FUNCTION_BLOCK INTERNAL FB_AlarmManager_Tests EXTENDS FB_TestSuite
VAR
	_dateTime	: ZigaLibs_Core.FB_LocalSystemTimeProvider;
	_alarmManager : FB_AlarmManager(
		enable := TRUE, // [BOOL] - Enables alarm generation
		logger := 0, // [REFERENCE TO ZigaLibs_Core.I_LoggerEx] - optional, logger.
		timeProvider := _dateTime); //[ZigaLibs_Core.I_LocalSystemTimeProvider] - required, date time provider.
END_VAR

_dateTime();
Test00_RegisterAlarms();
Test01_ActivateNewAlarm_ExpectUnacknowledgedActiveAlarm();
Test02_AcknowledgeActiveAlarm_ExpectActiveAcknowledged();
Test03_ActivateExistingAlarm_ExpectSameActiveAlarmCount();
Test04_DeactivateAlarm_ExpectNotActiveAcknowledged();
Test05_AcknowlidgeInactiveAlarm_ExpectAcknowledgedNotActive();
Test06_DisableManager_ExpectNoActiveAlarms();
Test07_AcknowledgeAllAlarms_ExpectActiveAlarmsUnchanged();
Test08_ActivateByName();
Test09_DeactivateByName();
Test10_AcknowledgeByName();
Test11_GetAlarmByName();
Test12_GetAlarmById();
Test13_ActivateById();
Test14_DeactivateById();
Test15_AcknowledgeById();
Test16_TimeInfos();
Test17_RaiseUnexisitngAlarm_ExpectNoNewAlarmsActive();
Test18_DeleteAlarm_ExpectPreviousAlarmsStillExist();
Test19_DeleteUnexistingAlarm_ExpectNoChangesToExistingAlarms();
Test20_DeleteAll();

METHOD Test00_RegisterAlarms
VAR_INPUT
END_VAR

VAR
	addAlarmIndex	: T_ArrayIndexer;
	alarm			: ST_AlarmInfo;
END_VAR
IF TcUnit.TEST_ORDERED('Test00_RegisterAlarms') THEN
	AssertEquals_UDINT(
		Actual := _alarmManager.RegisteredAlarmsCount,
		Expected := 0,
		Message := 'Before registering any alarms, the Registered count should be 0.');
	
	FOR addAlarmIndex := 1 TO 100 BY 1 DO
		AssertTrue(
			Condition := _alarmManager.RegisterAlarm(
				Id := addAlarmIndex,
				Message := Tc2_Standard.CONCAT('Alarm message', TO_STRING(addAlarmIndex)),
				Name := Tc2_Standard.CONCAT('Alarm name', TO_STRING(addAlarmIndex)),
				Level := E_AlarmLevel.INFO),
			Message := 'Registering alarm failed.');
			
		AssertEquals_UDINT(
			Actual := _alarmManager.RegisteredAlarmsCount,
			Expected := DINT_TO_UDINT(addAlarmIndex),
			Message := 'Registered alarm count is incorrect.');
			
		alarm := _alarmManager.GetAlarmById(nID := addAlarmIndex);
		AssertTrue(
			Condition := alarm.IsAcknowledged,
			Message := 'Newly registered alarm should be acknowledged by default, when created.');
	END_FOR
	
	AssertFalse(
		Condition := _alarmManager.RegisterAlarm(
			Id := 22,
			Message := CONCAT('Alarm message', TO_STRING(addAlarmIndex - 1)),
			Name := CONCAT('Alarm name', TO_STRING(addAlarmIndex - 1)),
			Level := E_AlarmLevel.INFO),
		Message := 'Registering an alarm with an existing id should not be possible.');
	
		
	TcUnit.TEST_FINISHED();
END_IF
END_METHOD

METHOD Test01_ActivateNewAlarm_ExpectUnacknowledgedActiveAlarm
VAR_INPUT
END_VAR

VAR
	currentAlarm	: ST_AlarmInfo;
END_VAR
IF TcUnit.TEST_ORDERED('Test01_ActivateNewAlarm_ExpectUnacknowledgedActiveAlarm') THEN
	_alarmManager.RaiseAlarmById(10);
	currentAlarm := _alarmManager.GetAlarmById(10);
	
	AssertEquals_BOOL(
		Actual := currentAlarm.IsActive,
		Expected := TRUE,
		Message := 'Alarm activation failed.');
		
	AssertEquals_BOOL(
		Actual := currentAlarm.IsAcknowledged,
		Expected := FALSE,
		Message := 'Newly activated alarm should not be acknowledged.');	
	
		
	AssertEquals_UINT(
		Actual := _alarmManager.ActiveAlarmsCount,
		Expected := 1,
		Message := 'Active alarm count is incorrect.');
	
	AssertEquals_UINT(
		Actual := _alarmManager.UnacknowledgedAlarmsCount,
		Expected := 1,
		Message := 'Unacknowledged alarm count is incorrect.');
		
	TcUnit.TEST_FINISHED();
END_IF
END_METHOD

METHOD Test02_AcknowledgeActiveAlarm_ExpectActiveAcknowledged
VAR_INPUT
END_VAR
IF TcUnit.TEST_ORDERED('Test02_AcknowledgeActiveAlarm_ExpectActiveAcknowledged') THEN

	_alarmManager.AcknowledgeAlarmById(10);
	
	AssertEquals_BOOL(
		Actual := _alarmManager.GetAlarmById(10).IsActive,
		Expected := TRUE,
		Message := 'Alarm activation failed.');
		
	AssertEquals_BOOL(
		Actual := _alarmManager.GetAlarmById(10).IsAcknowledged,
		Expected := TRUE,
		Message := 'Acknowlidging active alarm failed.');	
	
	TcUnit.TEST_FINISHED();
END_IF
END_METHOD

METHOD Test03_ActivateExistingAlarm_ExpectSameActiveAlarmCount
VAR_INPUT
END_VAR
IF TcUnit.TEST_ORDERED('Test03_ActivateExistingAlarm_ExpectSameActiveAlarmCount') THEN
	_alarmManager.RaiseAlarmById(10);	
	AssertEquals_BOOL(
		Actual := _alarmManager.GetAlarmById(10).IsActive,
		Expected := TRUE,
		Message := 'Alarm activation failed.');
		
	AssertEquals_BOOL(
		Actual := _alarmManager.GetAlarmById(10).IsAcknowledged,
		Expected := TRUE,
		Message := 'Already acknowledged alarm should not be acknowledged when activating the alarm while it is already active.');	
	
		
	AssertEquals_UINT(
		Actual := _alarmManager.ActiveAlarmsCount,
		Expected := 1,
		Message := 'Active alarm count is incorrect.');
	
	AssertEquals_UINT(
		Actual := _alarmManager.UnacknowledgedAlarmsCount,
		Expected := 0,
		Message := 'Activating acknowledged and already active alarm should not cause the alarm to be unacknowledged..');
		
	TcUnit.TEST_FINISHED();
END_IF
END_METHOD

METHOD Test04_DeactivateAlarm_ExpectNotActiveAcknowledged
VAR_INPUT
END_VAR
IF TcUnit.TEST_ORDERED('Test04_DeactivateAlarm_ExpectNotActiveAcknowledged') THEN
	_alarmManager.DeactivateAlarmById(10);
	
	AssertFalse(
		Condition := _alarmManager.GetAlarmById(10).IsActive,
		Message := 'Alarm deactivation failed.');
		
	AssertTrue(
		Condition := _alarmManager.GetAlarmById(10).IsAcknowledged,
		Message := 'Alarm deactivation should not acknowledge the alarm.');	
		
	AssertEquals_UINT(
		Actual := _alarmManager.ActiveAlarmsCount,
		Expected := 0,
		Message := 'Active alarm count is incorrect.');
	
	AssertEquals_UINT(
		Actual := _alarmManager.UnacknowledgedAlarmsCount,
		Expected := 0,
		Message := 'Unacknowledged alarm count is incorrect.');
		
	TcUnit.TEST_FINISHED();
END_IF
END_METHOD

METHOD Test05_AcknowlidgeInactiveAlarm_ExpectAcknowledgedNotActive
VAR_INPUT
END_VAR
IF TcUnit.TEST_ORDERED('Test05_AcknowlidgeInactiveAlarm_ExpectAcknowledgedNotActive') THEN
	_alarmManager.AcknowledgeAlarmById(10);
	
	AssertEquals_BOOL(
		Actual := _alarmManager.GetAlarmById(10).IsActive,
		Expected := FALSE,
		Message := 'Alarm deactivation failed.');
		
	AssertEquals_BOOL(
		Actual := _alarmManager.GetAlarmById(10).IsAcknowledged,
		Expected := TRUE,
		Message := 'Acknowlidging alarm failed.');	
	
		
	AssertEquals_UINT(
		Actual := _alarmManager.ActiveAlarmsCount,
		Expected := 0,
		Message := 'Active alarm count is incorrect.');
	
	AssertEquals_UINT(
		Actual := _alarmManager.UnacknowledgedAlarmsCount,
		Expected := 0,
		Message := 'Unacknowledged alarm count is incorrect.');
		
	TcUnit.TEST_FINISHED();
END_IF
END_METHOD

METHOD Test06_DisableManager_ExpectNoActiveAlarms
VAR_INPUT
END_VAR
VAR
	n	: T_ArrayIndexer;
END_VAR
IF TcUnit.TEST_ORDERED('Test06_DisableManager_ExpectNoActiveAlarms') THEN
	FOR n := 1 TO 40 BY 1 DO
		_alarmManager.RaiseAlarmById(n);
	END_FOR
	
	AssertEquals_UINT(
		Expected := 40,
		Actual := _alarmManager.ActiveAlarmsCount,
		Message := 'There should only be 40 active alarms at this point.');
			
	_alarmManager.Enable := FALSE;
	
	AssertEquals_UINT(
		Expected := 0,
		Actual := _alarmManager.ActiveAlarmsCount,
		Message := 'Disabling the manager should result in all of the alarms being inactive.');
	
	_alarmManager.Enable := TRUE;
	
	TcUnit.TEST_FINISHED();
END_IF
END_METHOD

METHOD Test07_AcknowledgeAllAlarms_ExpectActiveAlarmsUnchanged
VAR_INPUT
END_VAR

VAR
	n : T_ArrayIndexer;
	fbAlarmManager	: FB_AlarmManager(
		enable := TRUE, // [BOOL] - Enables alarm generation
		logger := 0, // [REFERENCE TO ZigaLibs_Core.I_LoggerEx] - optional, logger.
		timeProvider := _dateTime); //[ZigaLibs_Core.I_LocalSystemTimeProvider] - required, date time provider.
	arrAlarms		: ARRAY[0..60] OF ST_AlarmInfo;
END_VAR
IF TcUnit.TEST_ORDERED('Test07_AcknowledgeAllAlarms_ExpectActiveAlarmsUnchanged') THEN
	FOR n := 1 TO 40 BY 1 DO
		fbAlarmManager.RegisterAlarm(n, TO_STRING(n), '', E_AlarmLevel.INFO);
		fbAlarmManager.RaiseAlarmById(n);
	END_FOR
	
	AssertEquals_UINT(
		Expected := 40,
		Actual := fbAlarmManager.ActiveAlarmsCount,
		Message := 'There should only be 40 active alarms at this point.');
			
	fbAlarmManager.AcknowledgeAllAlarms();
	
	AssertEquals_UINT(
		Expected := 0,
		Actual := fbAlarmManager.UnacknowledgedAlarmsCount,
		Message := 'Acknowlidging all alarms should result in no unacknowledged alarms.');
	
	AssertEquals_UINT(
		Expected := 40,
		Actual := fbAlarmManager.ActiveAlarmsCount,
		Message := 'There should still be 40 active alarms, acknowlidning alarms should not affect alarm state.');
		
	TcUnit.TEST_FINISHED();
END_IF
END_METHOD

METHOD Test08_ActivateByName
VAR_INPUT
END_VAR
IF TcUnit.TEST_ORDERED('Test08_ActivateByName') THEN
	// Reset all alarms this way
	_alarmManager.Enable := FALSE;
	_alarmManager.Enable := TRUE;
	
	_alarmManager.RaiseAlarmByName('Alarm name10');
	
	AssertTrue(
		Condition := _alarmManager.GetAlarmByName('Alarm name10').IsActive,
		Message := 'Activating alarm by name failed.');
	
	AssertFalse(
		Condition := _alarmManager.GetAlarmByName('Alarm name10').IsAcknowledged,
		Message := 'Alarm shold be unacknowledged.');
		
	_alarmManager.DeactivateAlarmByName('Alarm name10');
	_alarmManager.AcknowledgeAlarmByName('Alarm name10');
	
	_alarmManager.Actions()
		.Raise()
		.ByName('Alarm name10');
	
	AssertTrue(
		Condition := _alarmManager.GetAlarmByName('Alarm name10').IsActive,
		Message := 'Fluent - Activating alarm by name failed.');
	
	AssertFalse(
		Condition := _alarmManager.GetAlarmByName('Alarm name10').IsAcknowledged,
		Message := 'Fluent - Alarm shold be unacknowledged.');
		
	TcUnit.TEST_FINISHED();
END_IF
END_METHOD

METHOD Test09_DeactivateByName
VAR_INPUT
END_VAR
IF TcUnit.TEST_ORDERED('Test09_DeactivateByName') THEN
	_alarmManager.DeactivateAlarmByName('Alarm name10');
	AssertFalse(
		Condition := _alarmManager.GetAlarmByName('Alarm name10').IsActive,
		Message := 'Deactivate alarm by name failed.');
	
	AssertFalse(
		Condition := _alarmManager.GetAlarmByName('Alarm name10').IsAcknowledged,
		Message := 'Alarm shold be unacknowledged.');
		
	_alarmManager.RaiseAlarmByName('Alarm name10');
		
	_alarmManager.Actions()
		.Deactivate()
		.ByName('Alarm name10');
	
	AssertFalse(
		Condition := _alarmManager.GetAlarmByName('Alarm name10').IsActive,
		Message := 'Fluent - deactivating alarm by name failed.');
	
	AssertFalse(
		Condition := _alarmManager.GetAlarmByName('Alarm name10').IsAcknowledged,
		Message := 'Fluent - Alarm shold be unacknowledged.');
		
	TcUnit.TEST_FINISHED();
END_IF
END_METHOD

METHOD Test10_AcknowledgeByName
VAR_INPUT
END_VAR
IF TcUnit.TEST_ORDERED('Test10_AcknowledgeByName') THEN
	_alarmManager.AcknowledgeAlarmByName('Alarm name10');
	
	AssertTrue(
		Condition := _alarmManager.GetAlarmByName('Alarm name10').IsAcknowledged,
		Message := 'Alarm shold be acknowledged.');
	
		
	_alarmManager.Actions().Raise().ByName('Alarm name10');
	_alarmManager.Actions().Deactivate().ByName('Alarm name10');
	_alarmManager.Actions().Acknowledge().ByName('Alarm name10');
	AssertTrue(
		Condition := _alarmManager.GetAlarmByName('Alarm name10').IsAcknowledged,
		Message := 'Fluent - Alarm shold be acknowledged.');
		
	TcUnit.TEST_FINISHED();
END_IF
END_METHOD

METHOD Test11_GetAlarmByName
VAR_INPUT
END_VAR

VAR_INST
	fbAlarmManager	: FB_AlarmManager(
		enable := TRUE, // [BOOL] - Enables alarm generation
		logger := 0, // [REFERENCE TO ZigaLibs_Core.I_LoggerEx] - optional, logger.
		timeProvider := _dateTime); //[ZigaLibs_Core.I_LocalSystemTimeProvider] - required, date time provider.
	i				: T_ArrayIndexer;
END_VAR
IF TcUnit.TEST_ORDERED('Test11_GetAlarmByName') THEN
	FOR i := 1 TO 11 BY 1 DO
		fbAlarmManager.RegisterAlarm(i, TO_STRING(i), '',E_AlarmLevel.INFO);
		AssertEquals_STRING(
			Actual := fbAlarmManager.GetAlarmByName(sName := TO_STRING(i)).Name,
			Expected := TO_STRING(i),
			Message := CONCAT('Getting alarm by name failed for alarm', TO_STRING(i)));	
	END_FOR
	
	AssertFalse(
		Condition := __ISVALIDREF(fbAlarmManager.GetAlarmByName('Surely I dont exist...')),
		Message := 'Fetching an alarm by non existing name should return invalid reference.');
	
	TcUnit.TEST_FINISHED();
END_IF
END_METHOD

METHOD Test12_GetAlarmById
VAR_INPUT
END_VAR
VAR_INST
	fbAlarmManager	: FB_AlarmManager(
		enable := TRUE, // [BOOL] - Enables alarm generation
		logger := 0, // [REFERENCE TO ZigaLibs_Core.I_LoggerEx] - optional, logger.
		timeProvider := _dateTime); //[ZigaLibs_Core.I_LocalSystemTimeProvider] - required, date time provider.
	i	: T_ArrayIndexer;
END_VAR
IF TcUnit.TEST_ORDERED('Test12_GetAlarmById') THEN
	FOR i := 1 TO 11 BY 1 DO
		fbAlarmManager.RegisterAlarm(i, TO_STRING(i), '', E_AlarmLevel.INFO);
		AssertEquals_DINT(
			Actual := fbAlarmManager.GetAlarmById(i).Id,
			Expected := i,
			Message := CONCAT('Getting alarm by id failed for alarm', TO_STRING(i)));	
	END_FOR
	
	TcUnit.TEST_FINISHED();
END_IF
END_METHOD

METHOD Test13_ActivateById
VAR_INPUT
END_VAR
IF TcUnit.TEST_ORDERED('Test13_ActivateById') THEN
	// Reset all alarms this way
	_alarmManager.Enable := FALSE;
	_alarmManager.Enable := TRUE;
	
	_alarmManager.RaiseAlarmById(10);
	
	AssertTrue(
		Condition := _alarmManager.GetAlarmById(10).IsActive,
		Message := 'Activating alarm by id failed.');
	
	AssertFalse(
		Condition := _alarmManager.GetAlarmById(10).IsAcknowledged,
		Message := 'Alarm shold be unacknowledged.');
		
	_alarmManager.DeactivateAlarmById(10);
	_alarmManager.AcknowledgeAlarmById(10);
	
	_alarmManager.Actions()
		.Raise()
		.ById(10);
	
	AssertTrue(
		Condition := _alarmManager.GetAlarmById(10).IsActive,
		Message := 'Fluent - Activating alarm by name failed.');
	
	AssertFalse(
		Condition := _alarmManager.GetAlarmById(10).IsAcknowledged,
		Message := 'Fluent - Alarm shold be unacknowledged.');
		
	TcUnit.TEST_FINISHED();
END_IF
END_METHOD

METHOD Test14_DeactivateById
VAR_INPUT
END_VAR
IF TcUnit.TEST_ORDERED('Test14_DeactivateById') THEN
	_alarmManager.DeactivateAlarmById(10);
	AssertFalse(
		Condition := _alarmManager.GetAlarmById(10).IsActive,
		Message := 'Deactivate alarm by name failed.');
	
	AssertFalse(
		Condition := _alarmManager.GetAlarmById(10).IsAcknowledged,
		Message := 'Alarm shold be unacknowledged.');
		
	_alarmManager.RaiseAlarmById(13);
		
	_alarmManager.Actions()
		.Deactivate()
		.ById(13);
	
	AssertFalse(
		Condition := _alarmManager.GetAlarmById(10).IsActive,
		Message := 'Fluent - deactivating alarm by name failed.');
	
	AssertFalse(
		Condition := _alarmManager.GetAlarmById(10).IsAcknowledged,
		Message := 'Fluent - Alarm shold be unacknowledged.');
		
	TcUnit.TEST_FINISHED();
END_IF
END_METHOD

METHOD Test15_AcknowledgeById
VAR_INPUT
END_VAR
IF TcUnit.TEST_ORDERED('Test15_AcknowledgeById') THEN
	_alarmManager.AcknowledgeAlarmById(10);
	
	AssertTrue(
		Condition := _alarmManager.GetAlarmById(10).IsAcknowledged,
		Message := 'Alarm shold be acknowledged.');
	
		
	_alarmManager.Actions().Raise().ById(10);
	_alarmManager.Actions().Deactivate().ById(10);
	_alarmManager.Actions().Acknowledge().ById(10);
	AssertTrue(
		Condition := _alarmManager.GetAlarmById(10).IsAcknowledged,
		Message := 'Fluent - Alarm shold be acknowledged.');
		
	TcUnit.TEST_FINISHED();
END_IF
END_METHOD

METHOD Test16_TimeInfos
VAR_INPUT
END_VAR

VAR_INST
	fbAlarmManager			: FB_AlarmManager(
		enable := TRUE, // [BOOL] - Enables alarm generation
		logger := 0, // [REFERENCE TO ZigaLibs_Core.I_LoggerEx] - optional, logger.
		timeProvider := _dateTime); //[ZigaLibs_Core.I_LocalSystemTimeProvider] - required, date time provider.
	i						: T_ArrayIndexer;
	stTimeStruct			: Tc2_Utilities.TIMESTRUCT;
	stTimeStructActivation	: Tc2_Utilities.TIMESTRUCT;	
	stTimeStructAcnowledge	: Tc2_Utilities.TIMESTRUCT;
	stTimeInfos	: ST_AlarmTimeInfos;
	alarm			: ST_AlarmInfo;
END_VAR
IF TcUnit.TEST_ORDERED('Test16_TimeInfos') THEN
	IF fbAlarmManager._dateTime.CurrentTime.IsValid THEN
		FOR i := 0 TO 10 BY 1 DO
			fbAlarmManager.RegisterAlarm(i,'','', E_AlarmLevel.INFO);
			
			IF NOT __ISVALIDREF(fbAlarmManager.GetAlarmById(i)) THEN
				AssertTrue(Condition := FALSE, 'Creating alarm failed, returned reference is invalid!');
			ELSE
				stTimeInfos := fbAlarmManager.GetAlarmById(i).TimeInfos;
			AssertEquals(
				Expected := stTimeStruct,
				Actual := fbAlarmManager.GetAlarmById(i).TimeInfos.Acknowledged,
				Message := 'Newly registered alarm should have empty TimeInfos.Acknowledged.');
			AssertEquals(
				Expected := stTimeStruct,
				Actual := fbAlarmManager.GetAlarmById(i).TimeInfos.Activated,
				Message := 'Newly registered alarm should have empty TimeInfos.Activated.');
			AssertEquals(
				Expected := stTimeStruct,
				Actual := fbAlarmManager.GetAlarmById(i).TimeInfos.Deactivated,
				Message := 'Newly registered alarm should have empty TimeInfos.Deactivated.');
			END_IF
		END_FOR
		
		// Raise alarm
		fbAlarmManager.Actions().Raise().ById(2);
		stTimeStruct := fbAlarmManager._dateTime.CurrentTime.Value;
		stTimeStructActivation := stTimeStruct;
		alarm := fbAlarmManager.GetAlarmById(2);
		AssertEquals_WORD(
			Expected := stTimeStruct.wMilliseconds,
			Actual := alarm.TimeInfos.Activated.wMilliseconds,
			Message := 'Activation time info after raising alarm (millisecond) is incorrect.');
		AssertEquals_WORD(
			Expected := stTimeStruct.wSecond,
			Actual := alarm.TimeInfos.Activated.wSecond,
			Message := 'Activation time info after raising alarm (second) is incorrect.');
		AssertEquals_WORD(
			Expected := stTimeStruct.wMinute,
			Actual := alarm.TimeInfos.Activated.wMinute,
			Message := 'Activation time info after raising alarm (minute) is incorrect.');
		AssertEquals_WORD(
			Expected := stTimeStruct.wHour,
			Actual := alarm.TimeInfos.Activated.wHour,
			Message := 'Activation time info after raising alarm (hour) is incorrect.');
		AssertEquals_WORD(
			Expected := stTimeStruct.wDay,
			Actual := alarm.TimeInfos.Activated.wDay,
			Message := 'Activation time info after raising alarm (day) is incorrect.');
		AssertEquals_WORD(
			Expected := stTimeStruct.wMonth,
			Actual := alarm.TimeInfos.Activated.wMonth,
			Message := 'Activation time info after raising alarm (month) is incorrect.');
		AssertEquals_WORD(
			Expected := stTimeStruct.wYear,
			Actual := alarm.TimeInfos.Activated.wYear,
			Message := 'Activation time info after raising alarm (year) is incorrect.');	
		AssertEquals_WORD(
			Expected := stTimeStruct.wDayOfWeek,
			Actual := alarm.TimeInfos.Activated.wDayOfWeek,
			Message := 'Activation time info after raising alarm (day of week) is incorrect.');
			
		MEMSET(ADR(stTimeStruct),0,SIZEOF(Tc2_Utilities.TIMESTRUCT));	
		AssertEquals(
			Expected := stTimeStruct,
			Actual := fbAlarmManager.GetAlarmById(2).TimeInfos.Acknowledged,
			Message := 'When alarm is raised, the acknowledged time information should be empty.');
		AssertEquals(
			Expected := stTimeStruct,
			Actual := fbAlarmManager.GetAlarmById(2).TimeInfos.Deactivated,
			Message := 'When alarm is raised, the deactivation time information should be empty.');
		
		// Acknowledge alarm
		fbAlarmManager.Actions().Acknowledge().ById(2);
		stTimeStruct := fbAlarmManager._dateTime.CurrentTime.Value;
		stTimeStructAcnowledge := stTimeStruct;
		alarm := fbAlarmManager.GetAlarmById(2);
		
		AssertEquals_WORD(
			Expected := stTimeStruct.wMilliseconds,
			Actual := alarm.TimeInfos.Acknowledged.wMilliseconds,
			Message := 'Acknowledged time info after acknowlidging alarm (millisecond) is incorrect.');
		AssertEquals_WORD(
			Expected := stTimeStruct.wSecond,
			Actual := alarm.TimeInfos.Acknowledged.wSecond,
			Message := 'Acknowledged time info after acknowlidging alarm (second) is incorrect.');
		AssertEquals_WORD(
			Expected := stTimeStruct.wMinute,
			Actual := alarm.TimeInfos.Acknowledged.wMinute,
			Message := 'Acknowledged time info after acknowlidging alarm (minute) is incorrect.');
		AssertEquals_WORD(
			Expected := stTimeStruct.wHour,
			Actual := alarm.TimeInfos.Acknowledged.wHour,
			Message := 'Acknowledged time info after acknowlidging alarm (hour) is incorrect.');
		AssertEquals_WORD(
			Expected := stTimeStruct.wDay,
			Actual := alarm.TimeInfos.Acknowledged.wDay,
			Message := 'Acknowledged time info after acknowlidging alarm (day) is incorrect.');
		AssertEquals_WORD(
			Expected := stTimeStruct.wMonth,
			Actual := alarm.TimeInfos.Acknowledged.wMonth,
			Message := 'Acknowledged time info after acknowlidging alarm (month) is incorrect.');
		AssertEquals_WORD(
			Expected := stTimeStruct.wYear,
			Actual := alarm.TimeInfos.Acknowledged.wYear,
			Message := 'Acknowledged time info after acknowlidging alarm (year) is incorrect.');	
		AssertEquals_WORD(
			Expected := stTimeStruct.wDayOfWeek,
			Actual := alarm.TimeInfos.Acknowledged.wDayOfWeek,
			Message := 'Acknowledged time info after acknowlidging alarm (day of week) is incorrect.');
		
		MEMSET(ADR(stTimeStruct),0,SIZEOF(Tc2_Utilities.TIMESTRUCT));	
		AssertEquals(
			Expected := stTimeStruct,
			Actual := fbAlarmManager.GetAlarmById(2).TimeInfos.Deactivated,
			Message := 'When alarm is acknowledged, the deactivation time information should not change.');
		AssertEquals(
			Actual := fbAlarmManager.GetAlarmById(2).TimeInfos.Activated,
			Expected := stTimeStructActivation,
			Message := 'If alarm is acknowledged, the acivation time info should not change.');
			
		// Deactivate alarm
		fbAlarmManager.Actions().Deactivate().ById(2);
		stTimeStruct := fbAlarmManager._dateTime.CurrentTime.Value;
		alarm := fbAlarmManager.GetAlarmById(2);
		
		AssertEquals_WORD(
			Expected := stTimeStruct.wMilliseconds,
			Actual := alarm.TimeInfos.Deactivated.wMilliseconds,
			Message := 'Deactivation time info after deactivating alarm (millisecond) is incorrect.');
		AssertEquals_WORD(
			Expected := stTimeStruct.wSecond,
			Actual := alarm.TimeInfos.Deactivated.wSecond,
			Message := 'Deactivation time info after deactivating alarm (second) is incorrect.');
		AssertEquals_WORD(
			Expected := stTimeStruct.wMinute,
			Actual := alarm.TimeInfos.Deactivated.wMinute,
			Message := 'Deactivation time info after deactivating alarm (minute) is incorrect.');
		AssertEquals_WORD(
			Expected := stTimeStruct.wHour,
			Actual := alarm.TimeInfos.Deactivated.wHour,
			Message := 'Deactivation time info after deactivating alarm (hour) is incorrect.');
		AssertEquals_WORD(
			Expected := stTimeStruct.wDay,
			Actual := alarm.TimeInfos.Deactivated.wDay,
			Message := 'Deactivation time info after deactivating alarm (day) is incorrect.');
		AssertEquals_WORD(
			Expected := stTimeStruct.wMonth,
			Actual := alarm.TimeInfos.Deactivated.wMonth,
			Message := 'Deactivation time info after deactivating alarm (month) is incorrect.');
		AssertEquals_WORD(
			Expected := stTimeStruct.wYear,
			Actual := alarm.TimeInfos.Deactivated.wYear,
			Message := 'Deactivation time info after deactivating alarm (year) is incorrect.');	
		AssertEquals_WORD(
			Expected := stTimeStruct.wDayOfWeek,
			Actual := alarm.TimeInfos.Deactivated.wDayOfWeek,
			Message := 'Deactivation time info after deactivating alarm (day of week) is incorrect.');
		
		// Check that previous entries did not change	
		AssertEquals(
			Expected := stTimeStructAcnowledge,
			Actual := fbAlarmManager.GetAlarmById(2).TimeInfos.Acknowledged,
			Message := 'When alarm is acknowledged, the deactivation time information should not change.');
		AssertEquals(
			Actual := fbAlarmManager.GetAlarmById(2).TimeInfos.Activated,
			Expected := stTimeStructActivation,
			Message := 'If alarm is acknowledged, the acivation time info should not change.');
		
			
		// Activate again and confirm that acknowledge and deactivation are reset
		// Raise alarm
		fbAlarmManager.Actions().Raise().ById(2);
		MEMSET(ADR(stTimeStruct),0,SIZEOF(Tc2_Utilities.TIMESTRUCT));
		AssertEquals(
			Actual := fbAlarmManager.GetAlarmById(2).TimeInfos.Deactivated,
			Expected := stTimeStruct,
			Message := 'When alarm is re-activated, previous time information for "deactivated" should be cleared.');
		AssertEquals(
			Actual := fbAlarmManager.GetAlarmById(2).TimeInfos.Acknowledged,
			Expected := stTimeStruct,
			Message := 'When alarm is re-activated, previous time information for "acknowledged" should be cleared.');
			
		TcUnit.TEST_FINISHED();
	END_IF
END_IF
END_METHOD

METHOD Test17_RaiseUnexisitngAlarm_ExpectNoNewAlarmsActive
VAR_INPUT
END_VAR

VAR_INST
	prevAlarmActiveCount	: UINT;
	prevUnackAlarmCount		: UINT;
END_VAR
IF TcUnit.TEST_ORDERED('Test17_RaiseUnexisitngAlarm_ExpectNoNewAlarmsActive') THEN
	prevAlarmActiveCount := _alarmManager.ActiveAlarmsCount;
	prevUnackAlarmCount := _alarmManager.UnacknowledgedAlarmsCount;
	
	_alarmManager.RaiseAlarmById(24523452);
	AssertEquals_UINT(
		Actual := _alarmManager.ActiveAlarmsCount,
		Expected := prevAlarmActiveCount,
		Message := 'If an alarm that does not exist is raised, active alarms count should not change.');
		
	AssertEquals_UINT(
		Actual := _alarmManager.UnacknowledgedAlarmsCount,
		Expected := prevUnackAlarmCount,
		Message := 'If an alarm that does not exist is raised, active alarms count should not change.');
		
	_alarmManager.Actions().Raise().ById(24523452);
	AssertEquals_UINT(
		Actual := _alarmManager.ActiveAlarmsCount,
		Expected := prevAlarmActiveCount,
		Message := 'Fluent - If an alarm that does not exist is raised, active alarms count should not change.');
		
	AssertEquals_UINT(
		Actual := _alarmManager.UnacknowledgedAlarmsCount,
		Expected := prevUnackAlarmCount,
		Message := 'Fluent - If an alarm that does not exist is raised, active alarms count should not change.');
		
	TcUnit.TEST_FINISHED();
END_IF
END_METHOD

METHOD Test18_DeleteAlarm_ExpectPreviousAlarmsStillExist
VAR_INPUT
END_VAR
VAR_INST
	fbAlarmManager	: FB_AlarmManager(
		enable := TRUE, // [BOOL] - Enables alarm generation
		logger := 0, // [REFERENCE TO ZigaLibs_Core.I_LoggerEx] - optional, logger.
		timeProvider := _dateTime); //[ZigaLibs_Core.I_LocalSystemTimeProvider] - required, date time provider.
	currentAlarm	: ST_AlarmInfo;
END_VAR
IF TcUnit.TEST_ORDERED('Test18_DeleteAlarm_ExpectPreviousAlarmsStillExist') THEN
	fbAlarmManager.RegisterAlarm(1,'1','1',E_AlarmLevel.WARNING);
	fbAlarmManager.RegisterAlarm(2,'2','2',E_AlarmLevel.WARNING);
	fbAlarmManager.RegisterAlarm(3,'3','3',E_AlarmLevel.WARNING);
	fbAlarmManager.RegisterAlarm(4,'4','4',E_AlarmLevel.WARNING);
	
	fbAlarmManager.DeleteAlarm(2);
	AssertEquals_UDINT(
		Expected := 3,
		Actual := fbAlarmManager.RegisteredAlarmsCount,
		Message := 'Deleting an alarm should lower registered alarms count.');
		
	// Alarm index 1	
	currentAlarm := fbAlarmManager.GetAlarmById(1);
	AssertEquals_DINT(
		Expected := 1,
		Actual := currentAlarm.Id,
		Message := 'First alarm Id is incorrected after deleting 2nd alarm.');
	AssertEquals_STRING(
		Expected := '1',
		Actual := currentAlarm.Name,
		Message := 'First alarm Name is incorrected after deleting 2nd alarm.');
	AssertEquals_STRING(
		Expected := '1',
		Actual := currentAlarm.Message,
		Message := 'First alarm Message is incorrected after deleting 2nd alarm.');
	
	// Alarm index 2	
	// Should no longer exist
	
	AssertFalse(
		Condition := __ISVALIDREF(fbAlarmManager.GetAlarmById(2)),
		Message := 'Alarm with Id 2 should no longer exist.');
	
	
	// Alarm index 3	
	AssertTrue(
			Condition := __ISVALIDREF(fbAlarmManager.GetAlarmById(3)),
			Message := 'Alarm with Id 3 should exist.');
			
	currentAlarm := fbAlarmManager.GetAlarmById(3);
	AssertEquals_DINT(
		Expected := 3,
		Actual := currentAlarm.Id,
		Message := '3rd alarm Id is incorrected after deleting 2nd alarm.');
	AssertEquals_STRING(
		Expected := '3',
		Actual := currentAlarm.Name,
		Message := '3rd alarm Name is incorrected after deleting 2nd alarm.');
	AssertEquals_STRING(
		Expected := '3',
		Actual := currentAlarm.Message,
		Message := '3rd alarm Message is incorrected after deleting 2nd alarm.');
		
	// Alarm index 4		
	currentAlarm := fbAlarmManager.GetAlarmById(4);
	AssertEquals_DINT(
		Expected := 4,
		Actual := currentAlarm.Id,
		Message := '4th alarm Id is incorrected after deleting 2nd alarm.');
	AssertEquals_STRING(
		Expected := '4',
		Actual := currentAlarm.Name,
		Message := '4th alarm Name is incorrected after deleting 2nd alarm.');
	AssertEquals_STRING(
		Expected := '4',
		Actual := currentAlarm.Message,
		Message := '4th alarm Message is incorrected after deleting 2nd alarm.');
		
	TcUnit.TEST_FINISHED();
END_IF
END_METHOD

METHOD Test19_DeleteUnexistingAlarm_ExpectNoChangesToExistingAlarms
VAR_INPUT
END_VAR
VAR_INST
	fbAlarmManager	: FB_AlarmManager(
		enable := TRUE, // [BOOL] - Enables alarm generation
		logger := 0, // [REFERENCE TO ZigaLibs_Core.I_LoggerEx] - optional, logger.
		timeProvider := _dateTime); //[ZigaLibs_Core.I_LocalSystemTimeProvider] - required, date time provider.
	currentAlarm	: ST_AlarmInfo;
	emptyAlarm		: ST_AlarmInfo;
END_VAR
IF TcUnit.TEST_ORDERED('Test19_DeleteUnexistingAlarm_ExpectNoChangesToExistingAlarms') THEN
	fbAlarmManager.RegisterAlarm(1,'1','1',E_AlarmLevel.ERROR);
	fbAlarmManager.RegisterAlarm(2,'2','2',E_AlarmLevel.INFO);
	fbAlarmManager.RegisterAlarm(3,'3','3',E_AlarmLevel.WARNING);
	fbAlarmManager.RegisterAlarm(4,'4','4',E_AlarmLevel.WARNING);
	
	// Delete unexisting alarm, expect no changes.
	fbAlarmManager.DeleteAlarm(0);
	AssertEquals_UDINT(
		Expected := 4,
		Actual := fbAlarmManager.RegisteredAlarmsCount,
		Message := 'Deleting unexisting alarm should not change registered alarms count.');
		
	currentAlarm := fbAlarmManager.GetAlarmById(1);
	AssertEquals_DINT(
		Expected := 1,
		Actual := currentAlarm.Id,
		Message := 'First alarm Id is incorrected after deleting unexisting alarm.');
	AssertEquals_STRING(
		Expected := '1',
		Actual := currentAlarm.Name,
		Message := 'First alarm Name is incorrected after deleting unexisting alarm.');
	AssertEquals_STRING(
		Expected := '1',
		Actual := currentAlarm.Message,
		Message := 'First alarm Message is incorrected after deleting unexisting alarm.');
		
	currentAlarm := fbAlarmManager.GetAlarmById(2);
	AssertEquals_DINT(
		Expected := 2,
		Actual := currentAlarm.Id,
		Message := '2nd alarm Id is incorrected after deleting unexisting alarm.');
	AssertEquals_STRING(
		Expected := '2',
		Actual := currentAlarm.Name,
		Message := '2nd alarm Name is incorrected after deleting unexisting alarm.');
	AssertEquals_STRING(
		Expected := '2',
		Actual := currentAlarm.Message,
		Message := '2nd alarm Message is incorrected after deleting unexisting alarm.');
		
	currentAlarm := fbAlarmManager.GetAlarmById(3);
	AssertEquals_DINT(
		Expected := 3,
		Actual := currentAlarm.Id,
		Message := '3rd alarm Id is incorrected after deleting unexisting alarm.');
	AssertEquals_STRING(
		Expected := '3',
		Actual := currentAlarm.Name,
		Message := '3rd alarm Name is incorrected after deleting unexisting alarm.');
	AssertEquals_STRING(
		Expected := '3',
		Actual := currentAlarm.Message,
		Message := '3rd alarm Message is incorrected after deleting unexisting alarm.');
		
	currentAlarm := fbAlarmManager.GetAlarmById(4);
	AssertEquals_DINT(
		Expected := 4,
		Actual := currentAlarm.Id,
		Message := '4th alarm Id is incorrected after deleting unexisting alarm.');
	AssertEquals_STRING(
		Expected := '4',
		Actual := currentAlarm.Name,
		Message := '4th alarm Name is incorrected after deleting unexisting alarm.');
	AssertEquals_STRING(
		Expected := '4',
		Actual := currentAlarm.Message,
		Message := '4th alarm Message is incorrected after deleting unexisting alarm.');
		
	TcUnit.TEST_FINISHED();
END_IF
END_METHOD

METHOD Test20_DeleteAll
VAR_INST
	fbAlarmManager	: FB_AlarmManager(
		enable := TRUE,
		logger := 0,
		timeProvider := _dateTime);
	currentAlarm
	: ST_AlarmInfo;
	emptyAlarm		: ST_AlarmInfo;
	i	: INT;
END_VAR
TcUnit.TEST('Test20_DeleteAll');

FOR i := 0 TO 5 BY 1 DO
	fbAlarmManager.RegisterAlarm(i, TO_STRING(i), TO_STRING(i), E_AlarmLevel.ERROR);
	fbAlarmManager.Actions().Raise().ById(i);
END_FOR

fbAlarmManager.DeleteAll();
AssertEquals_UDINT(0, fbAlarmManager.RegisteredAlarmsCount, 'Deleteing all alarms should result in the registered alarm count being 0.');
AssertEquals_DINT(0, fbAlarmMAnager.ActiveAlarmsCount, 'Deleting all alarms should result in active alarms count being 0');
AssertEquals_DINT(0, fbAlarmManager.UnacknowledgedAlarmsCount, 'Deleting all alarms should result in unacknowledged alarms count being 0');
AssertFalse(__ISVALIDREF(fbAlarmManager.GetAlarmById(1)), 'Attempting to retrive an alarm when they have all been deleted should return an empty reference.');

TcUnit.TEST_FINISHED();
END_METHOD

END_FUNCTION_BLOCK

(* stored: Version 1.1.0.1
   POU FB_AlarmManager_Tests: Id {10bfaa3e-65e7-0c01-2813-1ee946632c0a}, SpecialFunc None
   Method Test00_RegisterAlarms: Id {51a6cd53-1880-0584-2f70-df4bc0e86a21}
   Method Test01_ActivateNewAlarm_ExpectUnacknowledgedActiveAlarm: Id {7f0e9f4c-5bc2-0878-1385-3574e587c2ae}
   Method Test02_AcknowledgeActiveAlarm_ExpectActiveAcknowledged: Id {166cfe6f-deb4-0095-3098-ac602a6b90d2}
   Method Test03_ActivateExistingAlarm_ExpectSameActiveAlarmCount: Id {7965def8-d7ed-02d1-3b57-b23c8065de36}
   Method Test04_DeactivateAlarm_ExpectNotActiveAcknowledged: Id {96dcec83-f316-0d03-070c-713bf1d2bb41}
   Method Test05_AcknowlidgeInactiveAlarm_ExpectAcknowledgedNotActive: Id {beee53a0-3829-0e73-085d-3463db81918b}
   Method Test06_DisableManager_ExpectNoActiveAlarms: Id {b03481cc-e0d8-0ce1-3ecb-3abcdb72167d}
   Method Test07_AcknowledgeAllAlarms_ExpectActiveAlarmsUnchanged: Id {1a04ca75-ed21-0b83-3992-f864a8578b80}
   Method Test08_ActivateByName: Id {cb90bc6c-a663-0c9c-1b33-727dc3854afd}
   Method Test09_DeactivateByName: Id {99c997c1-4ac4-020e-34d2-567e99eb8a63}
   Method Test10_AcknowledgeByName: Id {153a742d-7155-0960-3ec2-022d030aac91}
   Method Test11_GetAlarmByName: Id {4d533791-6062-0bdf-2d13-a36fcb1dcdfe}
   Method Test12_GetAlarmById: Id {b2630015-c400-05d0-091b-055cd024cccf}
   Method Test13_ActivateById: Id {8d5ea681-fb36-0ca1-2731-31b329eb662b}
   Method Test14_DeactivateById: Id {fc5934bc-8eb0-0ffa-36ea-9b401169248a}
   Method Test15_AcknowledgeById: Id {c509bed5-546c-02a1-09cd-cec74a9aa394}
   Method Test16_TimeInfos: Id {655ee826-7aca-00ae-013d-246f4b134f0a}
   Method Test17_RaiseUnexisitngAlarm_ExpectNoNewAlarmsActive: Id {3b6b474e-0cb7-0914-0086-cb6760c65883}
   Method Test18_DeleteAlarm_ExpectPreviousAlarmsStillExist: Id {19be0180-cd2d-0235-0a07-8c2a1dad774c}
   Method Test19_DeleteUnexistingAlarm_ExpectNoChangesToExistingAlarms: Id {8902ea1c-3c82-000e-1006-87d3da5fe33c}
   Method Test20_DeleteAll: Id {43545f14-eb24-03df-2cad-4fdbe5ff7dcf} *)
